(* CoDeSys 2.3.9.59 project: PLC.pr6 *)
(* Libraries: STANDARD.LB6 *)

(* POU MAIN, LD *)
PROGRAM MAIN
VAR
	START AT %IX0.0: BOOL;
	STOP AT %IX0.1: BOOL;
	CONVEYOR AT %QX0.0: BOOL;
	WEIGHT AT %IW2: INT := 625;
	NUL AT %QX0.1: BOOL;
	NULV AT %QX0.2: BOOL;
	LENGTH: INT := 25;
	NULL: BOOL;
	WIDTH: INT := 10;
	NULW: BOOL;
	HEIGHT: INT := 5;
	NULH: BOOL;
	VOLUME: DINT;
	IS_URGENT AT %IX0.2: BOOL := 1;
	PINCODE AT %IW4: DINT := 380004;
	CITYCODE AT %QW6: DINT;
	AHMEDABAD AT %QX1.1: BOOL;
	SURAT AT %QX1.2: BOOL;
	RAJKOT AT %QX1.3: BOOL;
	JAMNAGAR AT %QX1.4: BOOL;
	DENSITY AT %QW14: DINT;

	LOW_D AT %QX2.0: BOOL;
	HIGH_D AT %QX2.1: BOOL;
	LIGHT AT %QX2.2: BOOL;
	MEDIUM AT %QX2.3: BOOL;
	HEAVY AT %QX2.4: BOOL;
	LCOUNT: CTU;
	RES: BOOL;
	LIGHT_COUNT: INT;
	MCOUNT: CTU;
	MEDIUM_COUNT: INT;
	HCOUNT: CTU;
	HEAVY_COUNT: INT;
	W_CHARGE AT %QW12: REAL;
	TOTAL_CHARGE AT %QW14: REAL;

	C_AHMEDABAD: CTU;
	AHMEDABAD_PARCEL: INT;
	C_SURAT: CTU;
	SURAT_PARCEL: INT;
	C_RAJKOT: CTU;
	RAJKOT_PARCEL: INT;
	C_JAMNAGAR: CTU;
	JAMNAGAR_PARCEL: INT;

	U_AHMEDABAD: CTU;
	AHMEDABAD_U_PARCEL: INT;
	U_SURAT: CTU;
	SURAT_U_PARCEL: INT;
	U_RAJKOT: CTU;
	RAJKOT_U_PARCEL: INT;
	U_JAMNAGAR: CTU;
	JAMNAGAR_U_PARCEL: INT;

	UAR:BOOL;
	UAY:BOOL;
	UAG:BOOL;
	CAR:BOOL;
	CAY:BOOL;
	CAG:BOOL;

	CRR:BOOL;
	CRY:BOOL;
	CRG:BOOL;
	URR:BOOL;
	URY:BOOL;
	URG:BOOL;

	CSR:BOOL;
	CSY:BOOL;
	CSG:BOOL;
	USR:BOOL;
	USY:BOOL;
	USG: BOOL;

	CJR:BOOL;
	CJY:BOOL;
	CJG:BOOL;
	UJR:BOOL;
	UJY:BOOL;
	UJG:BOOL;


	RCA: BOOL;

	T0: TON;
	T1: TON;
	T2: TON;
	T3: TON;
	RUA: BOOL;
	T4: TON;
	T5: TON;
	T6: TON;
	T7: TON;

	RUS: BOOL;
	RCS: BOOL;
	RUJ: BOOL;
	RCJ: BOOL;
	T14: TON;
	T15: TON;
	T12: TON;
	T13: TON;
	T10: TON;
	T11: TON;
	RUR: BOOL;
	RCR: BOOL;
	T8: TON;
	T9: TON;
	T17: TON;
	T16: TON;
	EVEN AT %QX2.5: BOOL;
	ODD AT %QX2.6: BOOL;

	UA AT %QX3.3: BOOL;
	UR AT %QX3.4: BOOL;
	US AT %QX3.5: BOOL;
	UJ AT %QX3.6: BOOL;

	CA AT %QX3.7: BOOL;
	RR AT %QX4.1: BOOL;
	CS AT %QX3.9: BOOL;
	CJ AT %QX2.9: BOOL;
	CMR AT %QX2.8: BOOL;
	LILA AT %QX0.6: BOOL;
	LAL AT %QX0.5: BOOL;
	PILA AT %QX0.4: BOOL;


	XXY: INT := 25;
	TOTAL: INT;
END_VAR
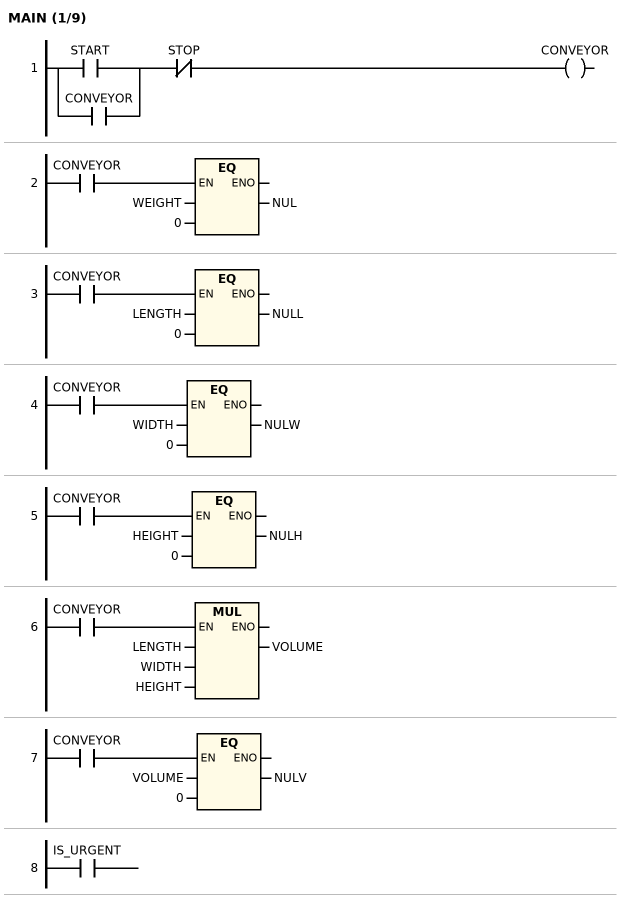
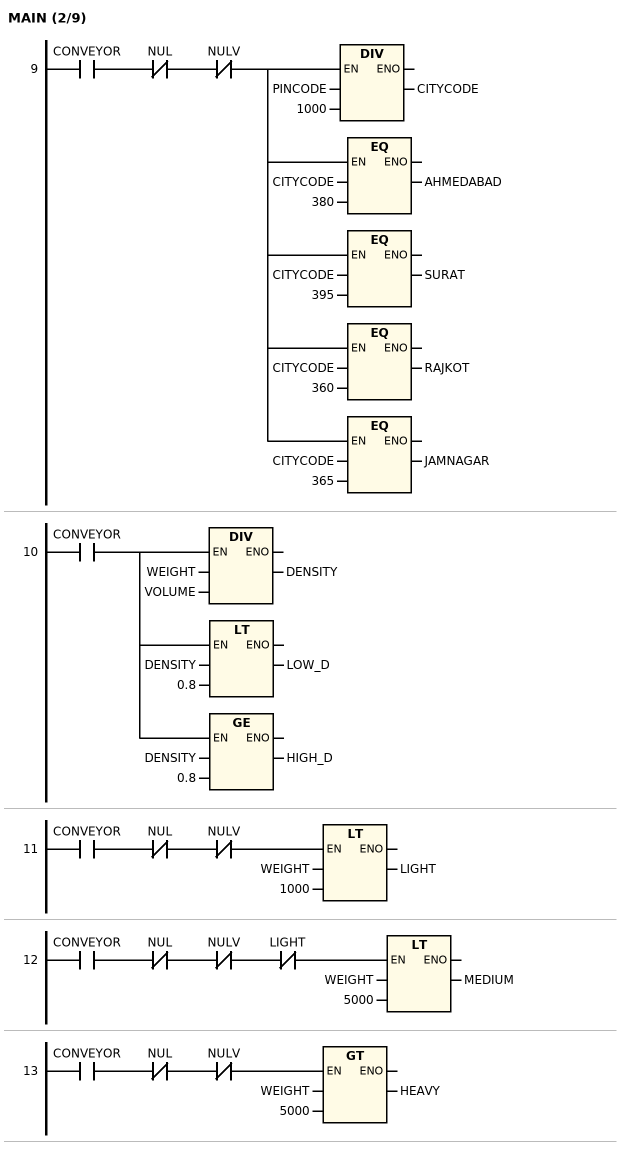
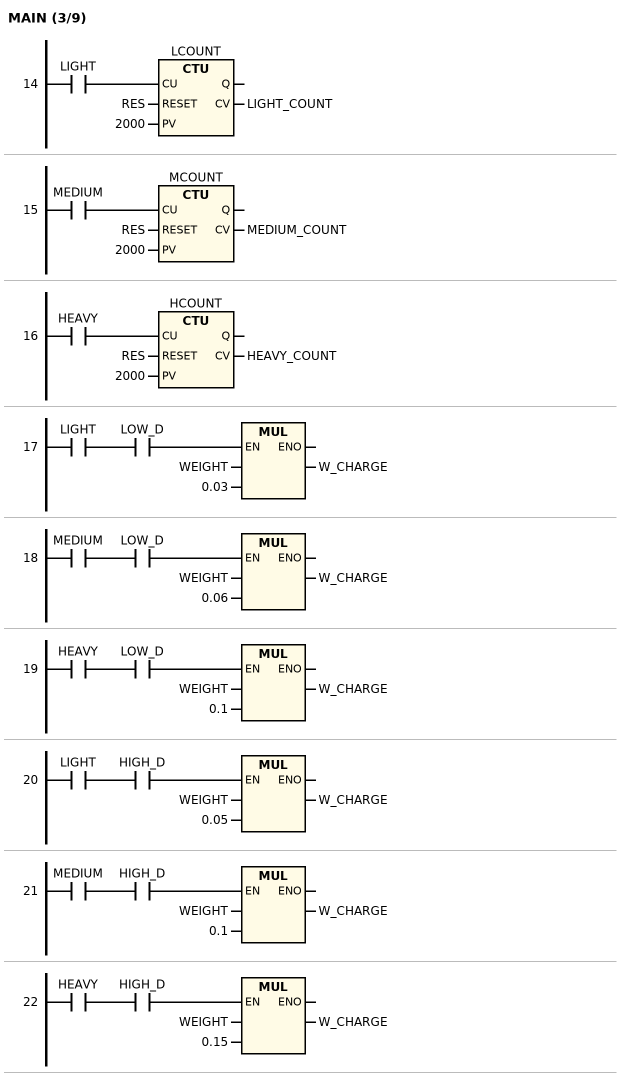
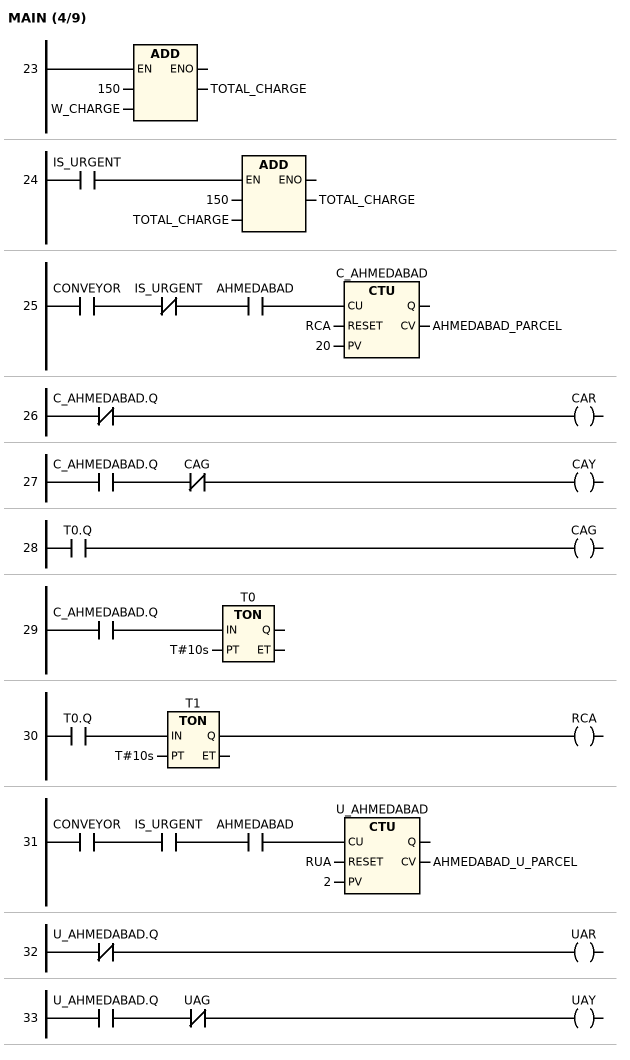
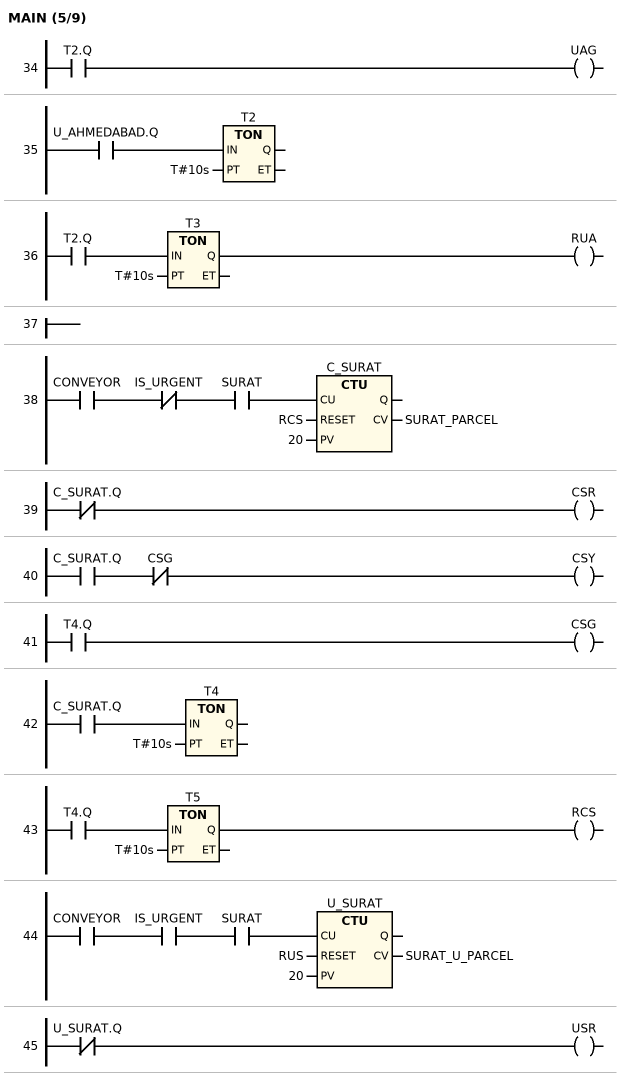
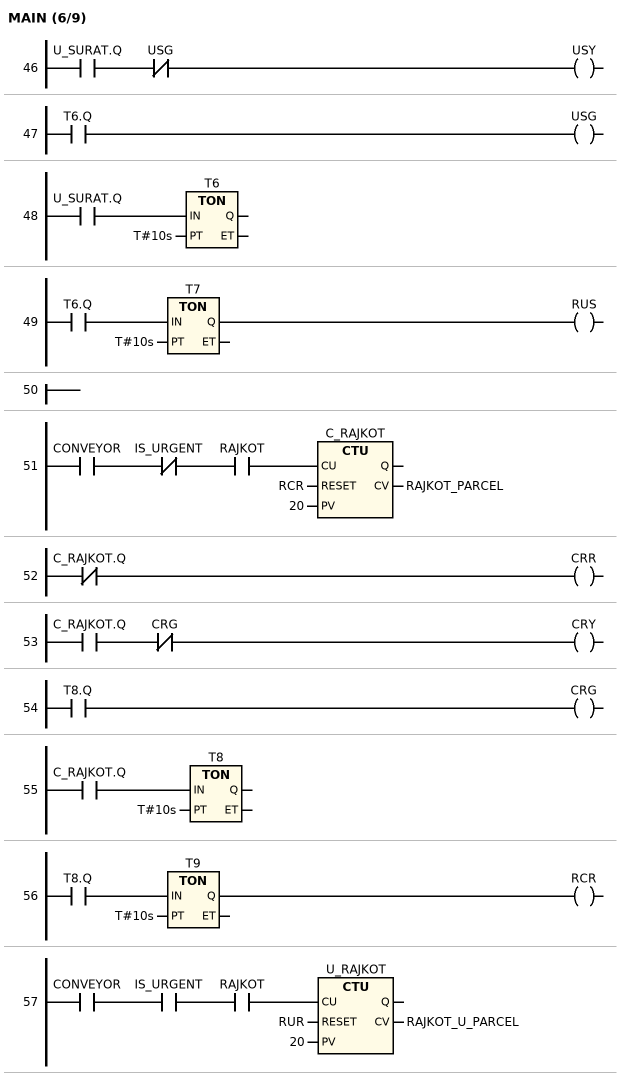
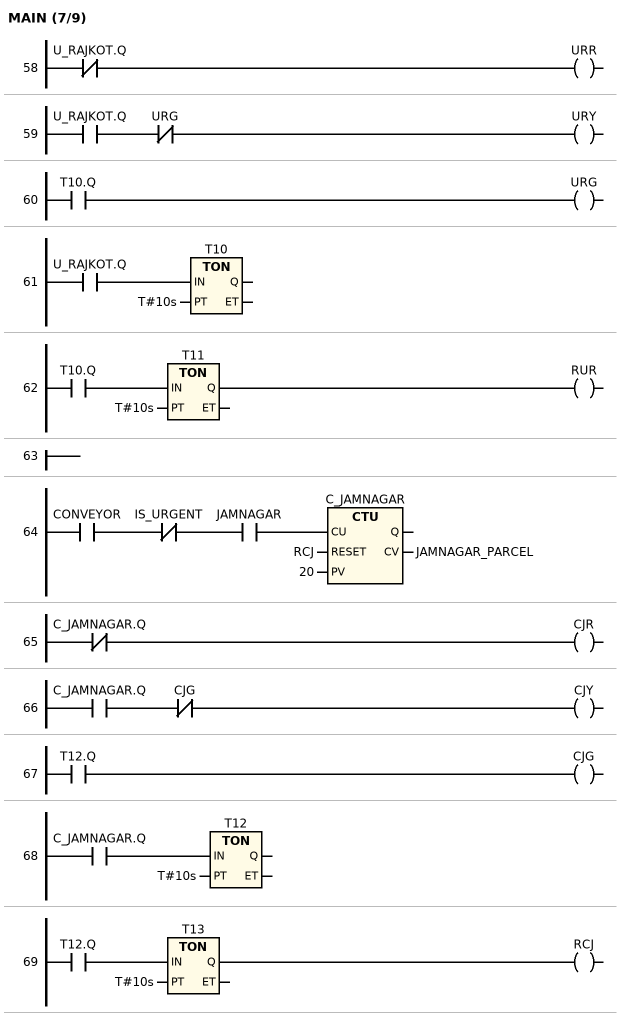
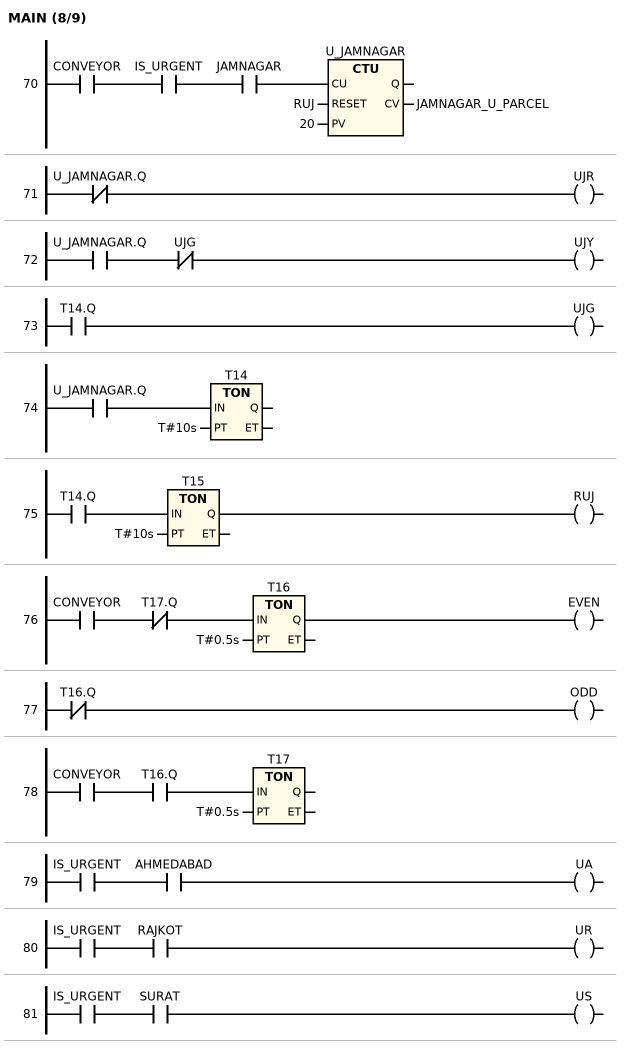
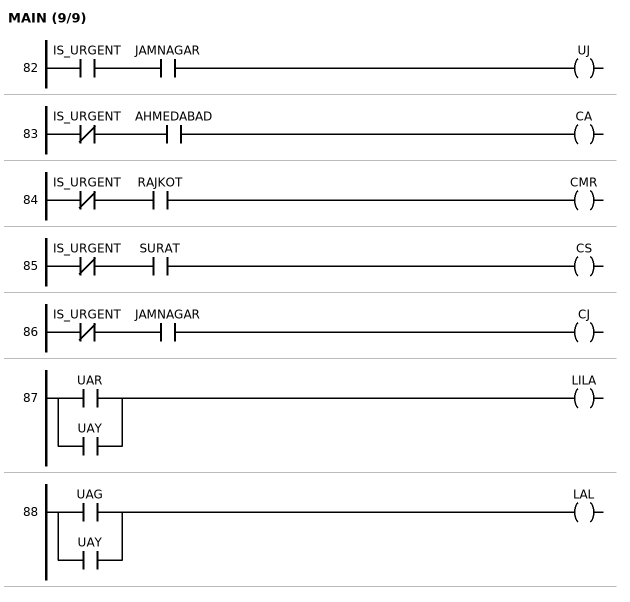
_LD_ (* Ladder Diagram *)
NETWORK 1
	{ [START] | [CONVEYOR] } - [/STOP] --- (CONVEYOR)
NETWORK 2
	[CONVEYOR]
		EN --- EQ(WEIGHT, 0) => NUL
NETWORK 3
	[CONVEYOR]
		EN --- EQ(LENGTH, 0) => NULL
NETWORK 4
	[CONVEYOR]
		EN --- EQ(WIDTH, 0) => NULW
NETWORK 5
	[CONVEYOR]
		EN --- EQ(HEIGHT, 0) => NULH
NETWORK 6
	[CONVEYOR]
		EN --- MUL(LENGTH, WIDTH, HEIGHT) => VOLUME
NETWORK 7
	[CONVEYOR]
		EN --- EQ(VOLUME, 0) => NULV
NETWORK 8
	[IS_URGENT]
NETWORK 9
	[CONVEYOR] - [/NUL] - [/NULV]
		EN --- DIV(PINCODE, 1000) => CITYCODE
		EN --- EQ(CITYCODE, 380) => AHMEDABAD
		EN --- EQ(CITYCODE, 395) => SURAT
		EN --- EQ(CITYCODE, 360) => RAJKOT
		EN --- EQ(CITYCODE, 365) => JAMNAGAR
NETWORK 10
	[CONVEYOR]
		EN --- DIV(WEIGHT, VOLUME) => DENSITY
		EN --- LT(DENSITY, 0.8) => LOW_D
		EN --- GE(DENSITY, 0.8) => HIGH_D
NETWORK 11
	[CONVEYOR] - [/NUL] - [/NULV]
		EN --- LT(WEIGHT, 1000) => LIGHT
NETWORK 12
	[CONVEYOR] - [/NUL] - [/NULV] - [/LIGHT]
		EN --- LT(WEIGHT, 5000) => MEDIUM
NETWORK 13
	[CONVEYOR] - [/NUL] - [/NULV]
		EN --- GT(WEIGHT, 5000) => HEAVY
NETWORK 14
	[LIGHT] - LCOUNT:CTU(CU: *, RESET: RES, PV: 2000, CV => LIGHT_COUNT)
NETWORK 15
	[MEDIUM] - MCOUNT:CTU(CU: *, RESET: RES, PV: 2000, CV => MEDIUM_COUNT)
NETWORK 16
	[HEAVY] - HCOUNT:CTU(CU: *, RESET: RES, PV: 2000, CV => HEAVY_COUNT)
NETWORK 17
	[LIGHT] - [LOW_D]
		EN --- MUL(WEIGHT, 0.03) => W_CHARGE
NETWORK 18
	[MEDIUM] - [LOW_D]
		EN --- MUL(WEIGHT, 0.06) => W_CHARGE
NETWORK 19
	[HEAVY] - [LOW_D]
		EN --- MUL(WEIGHT, 0.1) => W_CHARGE
NETWORK 20
	[LIGHT] - [HIGH_D]
		EN --- MUL(WEIGHT, 0.05) => W_CHARGE
NETWORK 21
	[MEDIUM] - [HIGH_D]
		EN --- MUL(WEIGHT, 0.1) => W_CHARGE
NETWORK 22
	[HEAVY] - [HIGH_D]
		EN --- MUL(WEIGHT, 0.15) => W_CHARGE
NETWORK 23
	*
		EN --- ADD(150, W_CHARGE) => TOTAL_CHARGE
NETWORK 24
	[IS_URGENT]
		EN --- ADD(150, TOTAL_CHARGE) => TOTAL_CHARGE
NETWORK 25
	[CONVEYOR] - [/IS_URGENT] - [AHMEDABAD] - C_AHMEDABAD:CTU(CU: *, RESET: RCA, PV: 20, CV => AHMEDABAD_PARCEL)
NETWORK 26
	[/C_AHMEDABAD.Q] --- (CAR)
NETWORK 27
	[C_AHMEDABAD.Q] - [/CAG] --- (CAY)
NETWORK 28
	[T0.Q] --- (CAG)
NETWORK 29
	[C_AHMEDABAD.Q] - T0:TON(IN: *, PT: T#10s)
NETWORK 30
	[T0.Q] - T1:TON(IN: *, PT: T#10s) --- (RCA)
NETWORK 31
	[CONVEYOR] - [IS_URGENT] - [AHMEDABAD] - U_AHMEDABAD:CTU(CU: *, RESET: RUA, PV: 2, CV => AHMEDABAD_U_PARCEL)
NETWORK 32
	[/U_AHMEDABAD.Q] --- (UAR)
NETWORK 33
	[U_AHMEDABAD.Q] - [/UAG] --- (UAY)
NETWORK 34
	[T2.Q] --- (UAG)
NETWORK 35
	[U_AHMEDABAD.Q] - T2:TON(IN: *, PT: T#10s)
NETWORK 36
	[T2.Q] - T3:TON(IN: *, PT: T#10s) --- (RUA)
NETWORK 37
	*
NETWORK 38
	[CONVEYOR] - [/IS_URGENT] - [SURAT] - C_SURAT:CTU(CU: *, RESET: RCS, PV: 20, CV => SURAT_PARCEL)
NETWORK 39
	[/C_SURAT.Q] --- (CSR)
NETWORK 40
	[C_SURAT.Q] - [/CSG] --- (CSY)
NETWORK 41
	[T4.Q] --- (CSG)
NETWORK 42
	[C_SURAT.Q] - T4:TON(IN: *, PT: T#10s)
NETWORK 43
	[T4.Q] - T5:TON(IN: *, PT: T#10s) --- (RCS)
NETWORK 44
	[CONVEYOR] - [IS_URGENT] - [SURAT] - U_SURAT:CTU(CU: *, RESET: RUS, PV: 20, CV => SURAT_U_PARCEL)
NETWORK 45
	[/U_SURAT.Q] --- (USR)
NETWORK 46
	[U_SURAT.Q] - [/USG] --- (USY)
NETWORK 47
	[T6.Q] --- (USG)
NETWORK 48
	[U_SURAT.Q] - T6:TON(IN: *, PT: T#10s)
NETWORK 49
	[T6.Q] - T7:TON(IN: *, PT: T#10s) --- (RUS)
NETWORK 50
	*
NETWORK 51
	[CONVEYOR] - [/IS_URGENT] - [RAJKOT] - C_RAJKOT:CTU(CU: *, RESET: RCR, PV: 20, CV => RAJKOT_PARCEL)
NETWORK 52
	[/C_RAJKOT.Q] --- (CRR)
NETWORK 53
	[C_RAJKOT.Q] - [/CRG] --- (CRY)
NETWORK 54
	[T8.Q] --- (CRG)
NETWORK 55
	[C_RAJKOT.Q] - T8:TON(IN: *, PT: T#10s)
NETWORK 56
	[T8.Q] - T9:TON(IN: *, PT: T#10s) --- (RCR)
NETWORK 57
	[CONVEYOR] - [IS_URGENT] - [RAJKOT] - U_RAJKOT:CTU(CU: *, RESET: RUR, PV: 20, CV => RAJKOT_U_PARCEL)
NETWORK 58
	[/U_RAJKOT.Q] --- (URR)
NETWORK 59
	[U_RAJKOT.Q] - [/URG] --- (URY)
NETWORK 60
	[T10.Q] --- (URG)
NETWORK 61
	[U_RAJKOT.Q] - T10:TON(IN: *, PT: T#10s)
NETWORK 62
	[T10.Q] - T11:TON(IN: *, PT: T#10s) --- (RUR)
NETWORK 63
	*
NETWORK 64
	[CONVEYOR] - [/IS_URGENT] - [JAMNAGAR] - C_JAMNAGAR:CTU(CU: *, RESET: RCJ, PV: 20, CV => JAMNAGAR_PARCEL)
NETWORK 65
	[/C_JAMNAGAR.Q] --- (CJR)
NETWORK 66
	[C_JAMNAGAR.Q] - [/CJG] --- (CJY)
NETWORK 67
	[T12.Q] --- (CJG)
NETWORK 68
	[C_JAMNAGAR.Q] - T12:TON(IN: *, PT: T#10s)
NETWORK 69
	[T12.Q] - T13:TON(IN: *, PT: T#10s) --- (RCJ)
NETWORK 70
	[CONVEYOR] - [IS_URGENT] - [JAMNAGAR] - U_JAMNAGAR:CTU(CU: *, RESET: RUJ, PV: 20, CV => JAMNAGAR_U_PARCEL)
NETWORK 71
	[/U_JAMNAGAR.Q] --- (UJR)
NETWORK 72
	[U_JAMNAGAR.Q] - [/UJG] --- (UJY)
NETWORK 73
	[T14.Q] --- (UJG)
NETWORK 74
	[U_JAMNAGAR.Q] - T14:TON(IN: *, PT: T#10s)
NETWORK 75
	[T14.Q] - T15:TON(IN: *, PT: T#10s) --- (RUJ)
NETWORK 76
	[CONVEYOR] - [/T17.Q] - T16:TON(IN: *, PT: T#0.5s) --- (EVEN)
NETWORK 77
	[/T16.Q] --- (ODD)
NETWORK 78
	[CONVEYOR] - [T16.Q] - T17:TON(IN: *, PT: T#0.5s)
NETWORK 79
	[IS_URGENT] - [AHMEDABAD] --- (UA)
NETWORK 80
	[IS_URGENT] - [RAJKOT] --- (UR)
NETWORK 81
	[IS_URGENT] - [SURAT] --- (US)
NETWORK 82
	[IS_URGENT] - [JAMNAGAR] --- (UJ)
NETWORK 83
	[/IS_URGENT] - [AHMEDABAD] --- (CA)
NETWORK 84
	[/IS_URGENT] - [RAJKOT] --- (CMR)
NETWORK 85
	[/IS_URGENT] - [SURAT] --- (CS)
NETWORK 86
	[/IS_URGENT] - [JAMNAGAR] --- (CJ)
NETWORK 87
	{ [UAR] | [UAY] } --- (LILA)
NETWORK 88
	{ [UAG] | [UAY] } --- (LAL)
_END_LD_
(* the same logic as Structured Text *)
(* Network 1 *)
CONVEYOR := (START OR CONVEYOR) AND NOT STOP;
(* Network 2 *)
IF CONVEYOR THEN
	NUL := WEIGHT = 0;
END_IF;
(* Network 3 *)
IF CONVEYOR THEN
	NULL := LENGTH = 0;
END_IF;
(* Network 4 *)
IF CONVEYOR THEN
	NULW := WIDTH = 0;
END_IF;
(* Network 5 *)
IF CONVEYOR THEN
	NULH := HEIGHT = 0;
END_IF;
(* Network 6 *)
IF CONVEYOR THEN
	VOLUME := LENGTH * WIDTH * HEIGHT;
END_IF;
(* Network 7 *)
IF CONVEYOR THEN
	NULV := VOLUME = 0;
END_IF;
(* Network 8 *)
(* Network 9 *)
IF CONVEYOR AND NOT NUL AND NOT NULV THEN
	CITYCODE := PINCODE / 1000;
	AHMEDABAD := CITYCODE = 380;
	SURAT := CITYCODE = 395;
	RAJKOT := CITYCODE = 360;
	JAMNAGAR := CITYCODE = 365;
END_IF;
(* Network 10 *)
IF CONVEYOR THEN
	DENSITY := WEIGHT / VOLUME;
	LOW_D := DENSITY < 0.8;
	HIGH_D := DENSITY >= 0.8;
END_IF;
(* Network 11 *)
IF CONVEYOR AND NOT NUL AND NOT NULV THEN
	LIGHT := WEIGHT < 1000;
END_IF;
(* Network 12 *)
IF CONVEYOR AND NOT NUL AND NOT NULV AND NOT LIGHT THEN
	MEDIUM := WEIGHT < 5000;
END_IF;
(* Network 13 *)
IF CONVEYOR AND NOT NUL AND NOT NULV THEN
	HEAVY := WEIGHT > 5000;
END_IF;
(* Network 14 *)
LCOUNT(CU := LIGHT, RESET := RES, PV := 2000);
LIGHT_COUNT := LCOUNT.CV;
(* Network 15 *)
MCOUNT(CU := MEDIUM, RESET := RES, PV := 2000);
MEDIUM_COUNT := MCOUNT.CV;
(* Network 16 *)
HCOUNT(CU := HEAVY, RESET := RES, PV := 2000);
HEAVY_COUNT := HCOUNT.CV;
(* Network 17 *)
IF LIGHT AND LOW_D THEN
	W_CHARGE := WEIGHT * 0.03;
END_IF;
(* Network 18 *)
IF MEDIUM AND LOW_D THEN
	W_CHARGE := WEIGHT * 0.06;
END_IF;
(* Network 19 *)
IF HEAVY AND LOW_D THEN
	W_CHARGE := WEIGHT * 0.1;
END_IF;
(* Network 20 *)
IF LIGHT AND HIGH_D THEN
	W_CHARGE := WEIGHT * 0.05;
END_IF;
(* Network 21 *)
IF MEDIUM AND HIGH_D THEN
	W_CHARGE := WEIGHT * 0.1;
END_IF;
(* Network 22 *)
IF HEAVY AND HIGH_D THEN
	W_CHARGE := WEIGHT * 0.15;
END_IF;
(* Network 23 *)
TOTAL_CHARGE := 150 + W_CHARGE;
(* Network 24 *)
IF IS_URGENT THEN
	TOTAL_CHARGE := 150 + TOTAL_CHARGE;
END_IF;
(* Network 25 *)
C_AHMEDABAD(CU := CONVEYOR AND NOT IS_URGENT AND AHMEDABAD, RESET := RCA, PV := 20);
AHMEDABAD_PARCEL := C_AHMEDABAD.CV;
(* Network 26 *)
CAR := NOT C_AHMEDABAD.Q;
(* Network 27 *)
CAY := C_AHMEDABAD.Q AND NOT CAG;
(* Network 28 *)
CAG := T0.Q;
(* Network 29 *)
T0(IN := C_AHMEDABAD.Q, PT := T#10s);
(* Network 30 *)
T1(IN := T0.Q, PT := T#10s);
RCA := T1.Q;
(* Network 31 *)
U_AHMEDABAD(CU := CONVEYOR AND IS_URGENT AND AHMEDABAD, RESET := RUA, PV := 2);
AHMEDABAD_U_PARCEL := U_AHMEDABAD.CV;
(* Network 32 *)
UAR := NOT U_AHMEDABAD.Q;
(* Network 33 *)
UAY := U_AHMEDABAD.Q AND NOT UAG;
(* Network 34 *)
UAG := T2.Q;
(* Network 35 *)
T2(IN := U_AHMEDABAD.Q, PT := T#10s);
(* Network 36 *)
T3(IN := T2.Q, PT := T#10s);
RUA := T3.Q;
(* Network 37 *)
(* Network 38 *)
C_SURAT(CU := CONVEYOR AND NOT IS_URGENT AND SURAT, RESET := RCS, PV := 20);
SURAT_PARCEL := C_SURAT.CV;
(* Network 39 *)
CSR := NOT C_SURAT.Q;
(* Network 40 *)
CSY := C_SURAT.Q AND NOT CSG;
(* Network 41 *)
CSG := T4.Q;
(* Network 42 *)
T4(IN := C_SURAT.Q, PT := T#10s);
(* Network 43 *)
T5(IN := T4.Q, PT := T#10s);
RCS := T5.Q;
(* Network 44 *)
U_SURAT(CU := CONVEYOR AND IS_URGENT AND SURAT, RESET := RUS, PV := 20);
SURAT_U_PARCEL := U_SURAT.CV;
(* Network 45 *)
USR := NOT U_SURAT.Q;
(* Network 46 *)
USY := U_SURAT.Q AND NOT USG;
(* Network 47 *)
USG := T6.Q;
(* Network 48 *)
T6(IN := U_SURAT.Q, PT := T#10s);
(* Network 49 *)
T7(IN := T6.Q, PT := T#10s);
RUS := T7.Q;
(* Network 50 *)
(* Network 51 *)
C_RAJKOT(CU := CONVEYOR AND NOT IS_URGENT AND RAJKOT, RESET := RCR, PV := 20);
RAJKOT_PARCEL := C_RAJKOT.CV;
(* Network 52 *)
CRR := NOT C_RAJKOT.Q;
(* Network 53 *)
CRY := C_RAJKOT.Q AND NOT CRG;
(* Network 54 *)
CRG := T8.Q;
(* Network 55 *)
T8(IN := C_RAJKOT.Q, PT := T#10s);
(* Network 56 *)
T9(IN := T8.Q, PT := T#10s);
RCR := T9.Q;
(* Network 57 *)
U_RAJKOT(CU := CONVEYOR AND IS_URGENT AND RAJKOT, RESET := RUR, PV := 20);
RAJKOT_U_PARCEL := U_RAJKOT.CV;
(* Network 58 *)
URR := NOT U_RAJKOT.Q;
(* Network 59 *)
URY := U_RAJKOT.Q AND NOT URG;
(* Network 60 *)
URG := T10.Q;
(* Network 61 *)
T10(IN := U_RAJKOT.Q, PT := T#10s);
(* Network 62 *)
T11(IN := T10.Q, PT := T#10s);
RUR := T11.Q;
(* Network 63 *)
(* Network 64 *)
C_JAMNAGAR(CU := CONVEYOR AND NOT IS_URGENT AND JAMNAGAR, RESET := RCJ, PV := 20);
JAMNAGAR_PARCEL := C_JAMNAGAR.CV;
(* Network 65 *)
CJR := NOT C_JAMNAGAR.Q;
(* Network 66 *)
CJY := C_JAMNAGAR.Q AND NOT CJG;
(* Network 67 *)
CJG := T12.Q;
(* Network 68 *)
T12(IN := C_JAMNAGAR.Q, PT := T#10s);
(* Network 69 *)
T13(IN := T12.Q, PT := T#10s);
RCJ := T13.Q;
(* Network 70 *)
U_JAMNAGAR(CU := CONVEYOR AND IS_URGENT AND JAMNAGAR, RESET := RUJ, PV := 20);
JAMNAGAR_U_PARCEL := U_JAMNAGAR.CV;
(* Network 71 *)
UJR := NOT U_JAMNAGAR.Q;
(* Network 72 *)
UJY := U_JAMNAGAR.Q AND NOT UJG;
(* Network 73 *)
UJG := T14.Q;
(* Network 74 *)
T14(IN := U_JAMNAGAR.Q, PT := T#10s);
(* Network 75 *)
T15(IN := T14.Q, PT := T#10s);
RUJ := T15.Q;
(* Network 76 *)
T16(IN := CONVEYOR AND NOT T17.Q, PT := T#0.5s);
EVEN := T16.Q;
(* Network 77 *)
ODD := NOT T16.Q;
(* Network 78 *)
T17(IN := CONVEYOR AND T16.Q, PT := T#0.5s);
(* Network 79 *)
UA := IS_URGENT AND AHMEDABAD;
(* Network 80 *)
UR := IS_URGENT AND RAJKOT;
(* Network 81 *)
US := IS_URGENT AND SURAT;
(* Network 82 *)
UJ := IS_URGENT AND JAMNAGAR;
(* Network 83 *)
CA := NOT IS_URGENT AND AHMEDABAD;
(* Network 84 *)
CMR := NOT IS_URGENT AND RAJKOT;
(* Network 85 *)
CS := NOT IS_URGENT AND SURAT;
(* Network 86 *)
CJ := NOT IS_URGENT AND JAMNAGAR;
(* Network 87 *)
LILA := UAR OR UAY;
(* Network 88 *)
LAL := UAG OR UAY;
END_PROGRAM

(* Visualisation VISUALIZATION
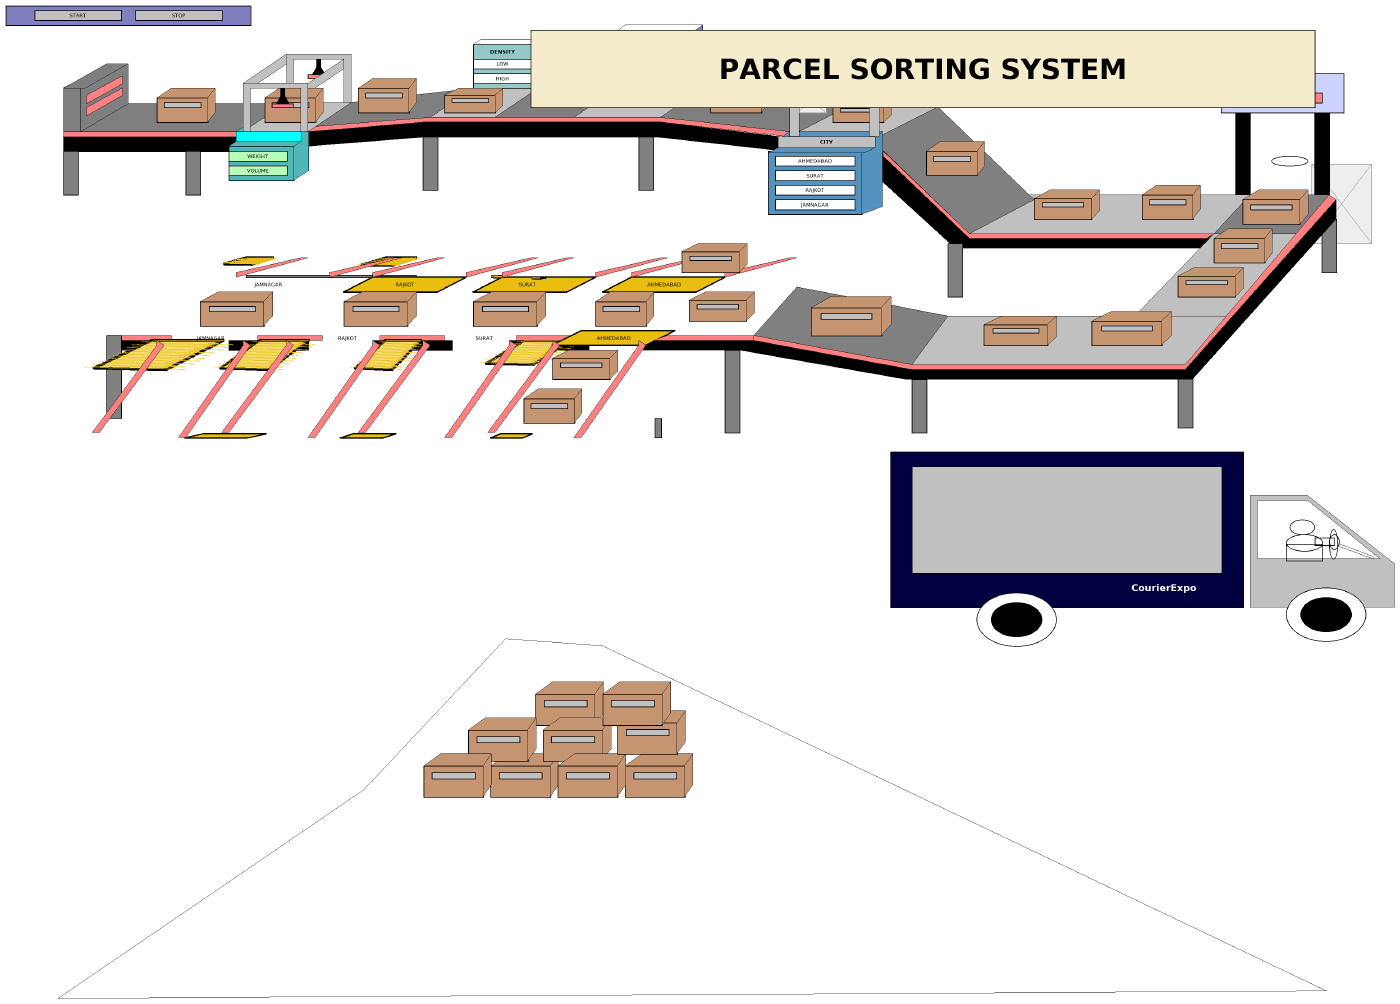
group at (260,300)-(2191,1681)
  bitmap at (1750,220)-(1831,331): c:\users\riddhi\onedrive\desktop\scan2.bmp
  group at (0,0)-(1861,891)
    polygon at (710,680)-(800,690): alarm colour if %QX0.0; toggles %QX0.0
    polygon at (520,680)-(610,690): alarm colour if %QX0.0; toggles %QX0.0
    polygon at (350,680)-(440,690): alarm colour if %QX0.0; toggles %QX0.0
    polygon at (140,680)-(230,690): alarm colour if %QX0.0; toggles %QX0.0
    group at (0,0)-(341,41)
      rectangle at (40,10)-(161,31): text "START"; alarm colour if %IX0.0; taps %IX0.0
      rectangle at (180,10)-(301,31): text "STOP"; alarm colour if %IX0.1; taps %IX0.1
    group at (650,70)-(751,171)
      rectangle at (0,40)-(81,61): text "LOW"; alarm colour if %QX2.0; toggles %QX2.0
      rectangle at (0,70)-(81,91): text "HIGH"; alarm colour if %QX2.1; toggles %QX2.1
      rectangle at (0,10)-(81,41): text "DENSITY"
    rectangle at (870,80)-(941,101): text "LIGHT"; alarm colour if %QX2.2; toggles %QX2.2
    rectangle at (870,140)-(941,161): text "HEAVY"; alarm colour if %QX2.4; toggles %QX2.4
    rectangle at (860,50)-(951,81): text "WEIGHT"
    rectangle at (870,110)-(941,131): text "MEDIUM"; alarm colour if %QX2.3; toggles %QX2.3
    rectangle at (1090,270)-(1201,301): text "CITY"
    rectangle at (1730,150)-(1801,171): text "URGENT"
    rectangle at (1710,180)-(1761,201): text "YES"; alarm colour if %IX0.2; toggles %IX0.2
    rectangle at (1780,180)-(1831,201): text "NO"; alarm colour if %IX0.2; toggles %IX0.2
    polygon at (80,260)-(320,280): alarm colour if %QX0.0; toggles %QX0.0
    polygon at (420,230)-(1090,270): alarm colour if %QX0.0; toggles %QX0.0
    ellipse at (1760,310)-(1811,331): alarm colour if %QX0.0; toggles %QX0.0
    bitmap at (1100,170)-(1141,221): c:\users\riddhi\onedrive\desktop\scan1.bmp
    bitmap at (1250,110)-(1291,161): c:\users\riddhi\onedrive\desktop\scan.bmp
    bitmap at (1180,110)-(1221,161): c:\users\riddhi\onedrive\desktop\scan.bmp
    rectangle at (1190,70)-(1281,101): text "BARCODE"
    polygon at (120,690)-(220,880): alarm colour if %QX3.6; toggles %QX3.6
    polygon at (240,690)-(340,890): alarm colour if %QX3.6; toggles %QX3.6
    polygon at (420,690)-(520,890): alarm colour if %QX3.4; toggles %QX3.4
    polygon at (610,690)-(710,890): alarm colour if %QX3.5; toggles %QX3.5
    polygon at (790,690)-(890,890): alarm colour if %QX3.3; toggles %QX3.3
    polygon at (300,690)-(400,880): alarm colour if %QX3.4; toggles %QX3.4
    polygon at (490,690)-(590,880): alarm colour if %QX3.5; toggles %QX3.5
    polygon at (670,690)-(770,880): alarm colour if %QX3.3; toggles %QX3.3
    rectangle at (800,670)-(891,701): text "AHMEDABAD"
    rectangle at (620,670)-(711,701): text "SURAT"
    rectangle at (430,670)-(521,701): text "RAJKOT"
    rectangle at (240,670)-(331,701): text "JAMNAGAR"
    rectangle at (870,560)-(961,591): text "AHMEDABAD"
    rectangle at (680,560)-(771,591): text "SURAT"
    rectangle at (510,560)-(601,591): text "RAJKOT"
    rectangle at (320,560)-(411,591): text "JAMNAGAR"
    polygon at (870,520)-(970,560): alarm colour if %QX3.7; toggles %QX3.7
    polygon at (1000,520)-(1100,560): alarm colour if %QX1.1; toggles %QX1.1
    polygon at (320,520)-(420,560): alarm colour if %QX2.9; toggles %QX2.9
    polygon at (450,520)-(550,560): alarm colour if %QX2.9; toggles %QX2.9
    polygon at (510,520)-(610,560): alarm colour if %QX3.8; toggles %QX3.8
    polygon at (640,520)-(740,560): alarm colour if %QX3.8; toggles %QX3.8
    polygon at (690,520)-(790,560): alarm colour if %QX3.9; toggles %QX3.9
    polygon at (820,520)-(920,560): alarm colour if %QX3.9; toggles %QX3.9
    polygon at (1220,300)-(1680,480): alarm colour if %QX0.0; toggles %QX0.0
    polygon at (900,680)-(1640,750): alarm colour if %QX0.0; toggles %QX0.0
    polygon at (1040,390)-(1850,750): alarm colour if %QX0.0; toggles %QX0.0
    rectangle at (1070,310)-(1181,331): text "AHMEDABAD"; alarm colour if %QX1.1; toggles %QX1.1
    polygon at (1074,270)-(1209,292): text "CITY"
    rectangle at (1070,340)-(1181,361): text "SURAT"; alarm colour if %QX1.2; toggles %QX1.2
    rectangle at (1070,370)-(1181,391): text "RAJKOT"; alarm colour if %QX1.3; toggles %QX1.3
    rectangle at (1070,400)-(1181,421): text "JAMNAGAR"; alarm colour if %QX1.4; toggles %QX1.4
    polygon at (112,144)-(162,202): alarm colour if %QX0.0; toggles %QX0.0
    polygon at (112,169)-(162,227): alarm colour if %QX0.0; toggles %QX0.0
    group at (420,110)-(450,151)
      rectangle at (0,32)-(30,41): alarm colour if %QX0.0; toggles %QX0.0
    group at (310,250)-(421,361)
      rectangle at (0,50)-(81,71): text "WEIGHT"; alarm colour if %QX0.1; toggles %QX0.1
      rectangle at (0,80)-(81,101): text "VOLUME"; alarm colour if %QX0.2; toggles %QX0.2
    group at (370,170)-(400,211)
      rectangle at (0,32)-(30,41): alarm colour if %QX0.0; toggles %QX0.0
    polygon at (1000,520)-(1100,560): alarm colour if %QX3.7; toggles %QX3.7
    group at (1230,920)-(1931,1321)
      rectangle at (30,30)-(461,251): invisible if %QX0.5
      rectangle at (30,30)-(461,251): invisible if %QX0.6
      rectangle at (270,240)-(491,321): text "CourierExpo"
    rectangle at (730,50)-(1821,211): text "PARCEL SORTING SYSTEM"
358 more shapes without text or variables
1 elements of other kinds (tables, trends, ...) not read
*)
